FUNCTION_BLOCK Idle IMPLEMENTS ITF_PackMLState, ITF_States
VAR
	_MyContext : ITF_PackMLMachine;
	_MyNextState : ITF_PackMLState;
	_MyStoppingState : ITF_PackMLState;
	_MyAbortingState : ITF_PackMLState;
END_VAR

PROPERTY AbortingState : ITF_PackMLState
GET
AbortingState := _MyAbortingState;
END_GET
SET
_MyAbortingState := AbortingState;
END_SET
END_PROPERTY

METHOD CyclicLogic : BOOL
VAR_INPUT
END_VAR
END_METHOD

{warning 'add method implementation '}
METHOD EStop : BOOL
END_METHOD

{warning 'add property implementation'}
PROPERTY MyNextState : ITF_PackMLState
GET
MyNextState := _MyNextState;
END_GET
SET
_MyNextState := MyNextState;
END_SET
END_PROPERTY

{warning 'add method implementation '}
METHOD Reset : BOOL
END_METHOD

{warning 'add method implementation '}
METHOD SetContext : BOOL
VAR_INPUT
	context	: ITF_PackMLMachine;
END_VAR
_MyContext := context;
END_METHOD

METHOD Start : BOOL
_MyContext.ChangeState(MyNextState);
END_METHOD

{warning 'add method implementation '}
METHOD Stop : BOOL
END_METHOD

{warning 'add property implementation'}
PROPERTY StoppingState : ITF_PackMLState
GET
StoppingState := _MyStoppingState;
END_GET
SET
_MyStoppingState := StoppingState;
END_SET
END_PROPERTY

END_FUNCTION_BLOCK

(* stored: Version 1.1.0.1, ProductVersion 3.1.4024.12
   POU Idle: Id {1a71340b-855d-47b4-8af3-2d3f122be3c4}, SpecialFunc None
   Property AbortingState: Id {16740356-b66c-4aa1-8a24-4e2d68686c88}
   Get Get: Id {fbea08cb-94b1-450b-9c8f-4e7f27de6a39}
   Set Set: Id {cd5556bf-fee8-42cc-ac6e-2435cc7a2845}
   Method CyclicLogic: Id {a5ec4d88-4540-415e-9a46-d7578f3cae61}
   Method EStop: Id {3f6dd750-e4c0-440d-b3f8-4473d8ce6b61}
   Property MyNextState: Id {1a2fa511-c9c8-4299-b4dc-b88cc8710b13}
   Get Get: Id {f2718f7e-5237-482a-80bd-91d1188975d7}
   Set Set: Id {5268af1d-e3fe-43b6-8b01-38f1c1aa0c1c}
   Method Reset: Id {8c045b4a-999b-4563-8473-bd3ae698008d}
   Method SetContext: Id {dfa932ae-f2e7-4f87-b5e6-d23722c940bb}
   Method Start: Id {34ca202e-52e0-4fbc-9e00-d3f29dfcabcb}
   Method Stop: Id {5bdd16e5-bc26-4e93-ae5f-93d096ef6a87}
   Property StoppingState: Id {77dd7774-d7f6-4dc4-8271-f9f973ebfd23}
   Get Get: Id {74ca09e6-e0cb-4aed-8f02-f1a1acae8b7d}
   Set Set: Id {80ffdc44-ecd7-43d8-a312-25d25c798910} *)
